TYPE OsSta_MB_V1 :
   STRUCT
      BX : Bool;
      Y : Bool;
      Alarm : Bool;
      Warning : Bool;
      Fault : Bool;
      Latched : Bool;
      Blocked : Bool;
      Suppressed : Bool;
      ForcedBlocked : Bool;
      ForcedSuppressed : Bool;
   END_STRUCT
END_TYPE

(* stored: Version 1.1.0.1, ProductVersion 3.1.4024.12
   DUT OsSta_MB_V1: Id {572155cd-1cb7-4296-b8e0-698682541d76} *)
